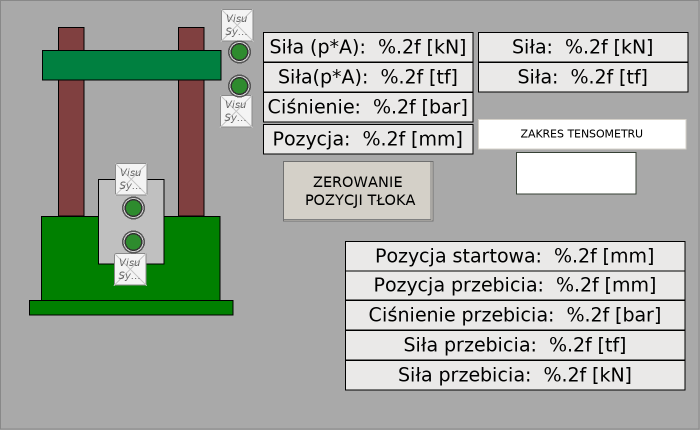
VISUALIZATION E0  // 700x430
    Textfield (263,92 210x30), "Ciśnienie: %.2f [bar]", text variable: Scaling.PressureAI.PV_Value
    Textfield (263,124 210x30), "Pozycja: %.2f [mm]", text variable: Scaling.fbPos.PosZeroed_mm
    Textfield (345,300 340x30), "Ciśnienie przebicia: %.2f [bar]", text variable: GVL_HMI.nPressBreak
    Textfield (345,270 340x30), "Pozycja przebicia: %.2f [mm]", text variable: GVL_HMI.nPositionBreak
    Textfield (345,241 340x30), "Pozycja startowa: %.2f [mm]", text variable: GVL_HMI.nPositionStart
    Rectangle (58,27 26x189)
    Rectangle (178,27 26x189)
    Rectangle (41,216 179x85)
    Rectangle (98,179 66x85)
    Rectangle (42,50 179x30)
    Group (220,9 35x118)
        Group (1,0 34x56)
            Image (0,0 32x32), colour toggle: bTopPreserUp, image: VisuSymbols.Symbols.ArrowBoldUp
            Lamp1 (3,30 31x26), variable: bTopPreserDown, style: Lamp-Lamp1-Green
        Group (0,64 35x54)
            Image (0,22 32x32), image: VisuSymbols.Symbols.ArrowBoldDown
            Lamp1 (4,0 31x26), variable: bTopPreserUp, style: Lamp-Lamp1-Green
    Group (114,163 35x122)
        Group (1,0 34x58)
            Image (0,0 32x32), colour toggle: bCylinderValveUp, image: VisuSymbols.Symbols.ArrowBoldUp
            Lamp1 (3,32 31x26), variable: bCylinderValveUp, style: Lamp-Lamp1-Green
        Group (0,66 35x56)
            Image (0,24 32x32), colour toggle: bCylinderValveDown, image: VisuSymbols.Symbols.ArrowBoldDown
            Lamp1 (4,0 31x26), variable: bCylinderValveDown, style: Lamp-Lamp1-Green
    Textfield (263,62 210x30), "Siła(p*A): %.2f [tf]", text variable: GVL_HMI.Force_kg/1000
    Textfield (263,32 210x30), "Siła (p*A): %.2f [kN]", text variable: GVL_HMI.Force_N/1000
    Rectangle (29,300 204x15)
    Textfield (478,62 210x30), "Siła: %.2f [tf]", text variable: GVL_ForceMode.nForce_t
    Textfield (478,32 210x30), "Siła: %.2f [kN]", text variable: GVL_ForceMode.nForce_kN
    Rectangle (516,152 120x42), colour toggle: P_EventsVisu.bFilterActiveOnly, input disabled if: bLedCycleOn, text list: 'Tensometr', text index: GVL_ForceMode.bForceRange100t
        toggle GVL_ForceMode.bForceRange100t
    Textfield (345,330 340x30), "Siła przebicia: %.2f [tf]", text variable: GVL_HMI.nForce_t_Break
    Textfield (345,360 340x30), "Siła przebicia: %.2f [kN]", text variable: GVL_HMI.nForce_kN_Break
    Textfield (478,119 208x30), "ZAKRES TENSOMETRU"
    Button (283,161 150x60), "ZEROWANIE POZYCJI TŁOKA", input disabled if: bLedCycleOn
        OnMouseDown: execute { Scaling.fbPos.SetZero:=false; }
        OnMouseUp: execute { Scaling.fbPos.SetZero:=true; }
END_VISUALIZATION

(* stored: Version 1.1.0.1, ProductVersion 3.1.4024.16
   Visu E0: Id {f3f1301d-3a4c-4a61-b2b4-31f212846622} *)
